{attribute 'qualified_only'}
{attribute 'strict'}
TYPE StateHeat :
(
	Off,
	Init,
	Ready,
	Heat,
	Hold,
	Done
);
END_TYPE

(* stored: Version 1.1.0.1, ProductVersion 3.1.4024.6
   DUT StateHeat: Id {b1b7830b-c383-4a2d-a887-74caea0600ba} *)
